INTERFACE ITF_0_BaseComponent

METHOD Activate : BOOL
VAR_INPUT
END_VAR
END_METHOD

METHOD Cleanup : BOOL
VAR_INPUT
END_VAR
END_METHOD

METHOD Configure : BOOL
VAR_INPUT
END_VAR
END_METHOD

METHOD Deactivate : BOOL
VAR_INPUT
END_VAR
END_METHOD

METHOD Destroy : BOOL
VAR_INPUT
END_VAR
END_METHOD

PROPERTY ID : UINT
GET
END_GET
SET
END_SET
END_PROPERTY

PROPERTY Name : String
GET
END_GET
END_PROPERTY

PROPERTY Path : String
GET
END_GET
END_PROPERTY

METHOD Shutdown : BOOL
VAR_INPUT
END_VAR
END_METHOD

PROPERTY ABSTRACT State : eState
GET
END_GET
SET
END_SET
END_PROPERTY

END_INTERFACE

(* stored: Version 1.1.0.1, ProductVersion 3.1.4026.18
   Itf ITF_0_BaseComponent: Id {65885d39-4024-4344-a8ab-374a6ccc4c59}
   Folder Transitions: Id {6560e606-0171-480a-9918-20910c0e5bdf}
   Method Activate: Id {421c2108-8179-4a12-ba41-35989c996212}
   Method Cleanup: Id {2b58a7de-95d9-467c-85d1-db9dec921482}
   Method Configure: Id {e50a6f49-0903-48ba-8271-1c9d1e1e510c}
   Method Deactivate: Id {543d663f-3433-4738-bb10-46e710584fb3}
   Method Destroy: Id {8dc262df-163a-4e11-9777-3fbb1a531627}
   Property ID: Id {fc62148d-d821-4a08-a5bf-6bdef92d59d5}
   Get Get: Id {c2985394-0d19-4b0e-a4c8-339d4db8e630}
   Set Set: Id {98424317-6db3-4da6-80d9-cb32dfe7d9a6}
   Property Name: Id {8e02e470-71da-44a6-a68f-092954d86151}
   Get Get: Id {7f1ff7dd-a478-4f29-885d-9677ae5d4a7e}
   Property Path: Id {755b1bdf-ea5e-45d8-b845-25d127de2ac2}
   Get Get: Id {bdac12b3-22bb-41f6-8039-bf0761521d8e}
   Method Shutdown: Id {d44b7757-327e-4329-96cc-8c180a9fb4f3}
   Property State: Id {4c5eddbd-3571-4017-85b4-cee88242beba}
   Get Get: Id {42aa47ea-f1d7-4040-ade8-b3efc7baaa84}
   Set Set: Id {1f4e04c9-7da1-43ff-a8c5-ecbad9f49fcd} *)
